// SIMATIC STEP 7 (V5.x) project PRACTICAS MOV-E
// CPU: CPU313 C-2 DP(1)
// station: P_ADR_BUS
// station: Hardware
// station: Equipo SIMATIC 300
// program: Programa S7(1)

SYMBOL_TABLE
"FLANCOS"	DB 1	DB 1
"P MARCHA"	I 0.0	BOOL
"P PARO"	I 0.1	BOOL
"Cycle Execution"	OB 1	OB 1
END_SYMBOL_TABLE

DATA_BLOCK "FLANCOS"	// DB 1
VERSION : 0.1
  STRUCT
   M0 : BOOL ;
   M1 : BOOL ;
   M2 : BOOL ;
   M3 : BOOL ;
   M4 : BOOL ;
   M5 : BOOL ;
   M6 : BOOL ;
   M7 : BOOL ;
  END_STRUCT ;	
BEGIN
END_DATA_BLOCK

ORGANIZATION_BLOCK "Cycle Execution"	// OB 1
TITLE = "Main Program Sweep (Cycle)"
VERSION : 0.1
VAR_TEMP
  OB1_EV_CLASS : BYTE ;	//Bits 0-3 = 1 (Coming event), Bits 4-7 = 1 (Event class 1)
  OB1_SCAN_1 : BYTE ;	//1 (Cold restart scan 1 of OB 1), 3 (Scan 2-n of OB 1)
  OB1_PRIORITY : BYTE ;	//Priority of OB Execution
  OB1_OB_NUMBR : BYTE ;	//1 (Organization block 1, OB1)
  OB1_RESERVED_1 : BYTE ;	//Reserved for system
  OB1_RESERVED_2 : BYTE ;	//Reserved for system
  OB1_PREV_CYCLE : INT ;	//Cycle time of previous OB1 scan (milliseconds)
  OB1_MIN_CYCLE : INT ;	//Minimum cycle time of OB1 (milliseconds)
  OB1_MAX_CYCLE : INT ;	//Maximum cycle time of OB1 (milliseconds)
  OB1_DATE_TIME : DATE_AND_TIME ;	//Date and time OB1 started
END_VAR
BEGIN
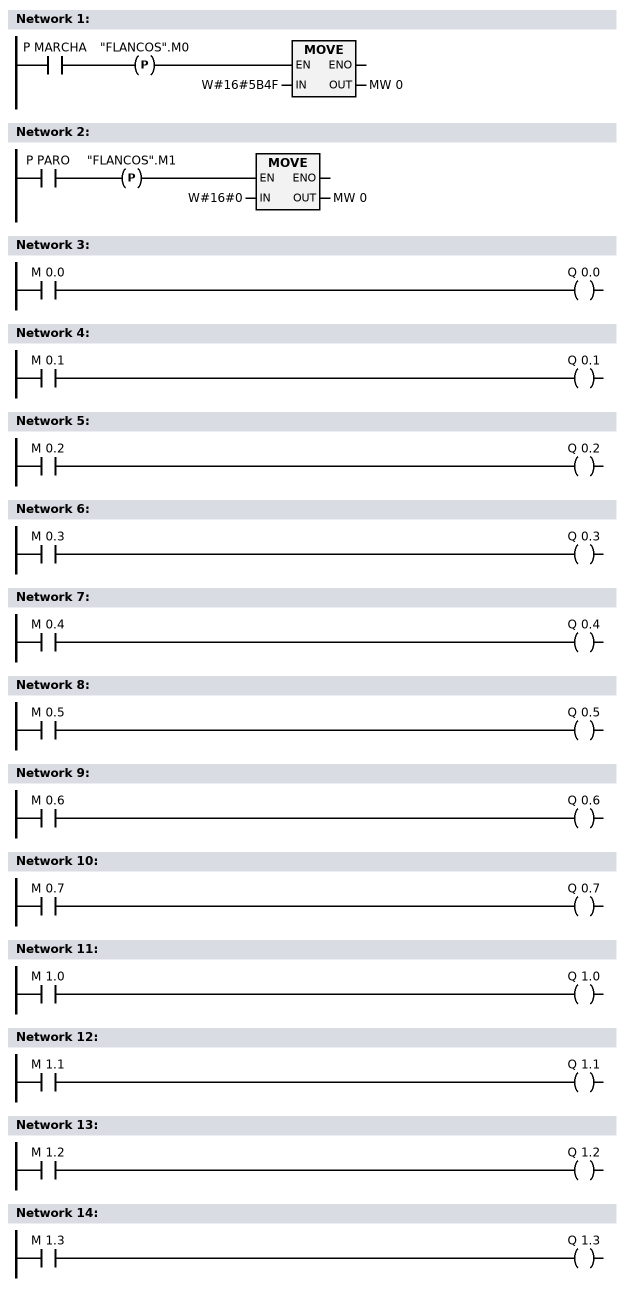
NETWORK
TITLE =
      A     "P MARCHA";
      FP    "FLANCOS".M0;
      JNB   _001;
      L     W#16#5B4F;
      T     MW 0;
_001: NOP   0;
NETWORK
TITLE =
      A     "P PARO";
      FP    "FLANCOS".M1;
      JNB   _002;
      L     W#16#0;
      T     MW 0;
_002: NOP   0;
NETWORK
TITLE =
      A     M 0.0;
      =     Q 0.0;
NETWORK
TITLE =
      A     M 0.1;
      =     Q 0.1;
NETWORK
TITLE =
      A     M 0.2;
      =     Q 0.2;
NETWORK
TITLE =
      A     M 0.3;
      =     Q 0.3;
NETWORK
TITLE =
      A     M 0.4;
      =     Q 0.4;
NETWORK
TITLE =
      A     M 0.5;
      =     Q 0.5;
NETWORK
TITLE =
      A     M 0.6;
      =     Q 0.6;
NETWORK
TITLE =
      A     M 0.7;
      =     Q 0.7;
NETWORK
TITLE =
      A     M 1.0;
      =     Q 1.0;
NETWORK
TITLE =
      A     M 1.1;
      =     Q 1.1;
NETWORK
TITLE =
      A     M 1.2;
      =     Q 1.2;
NETWORK
TITLE =
      A     M 1.3;
      =     Q 1.3;
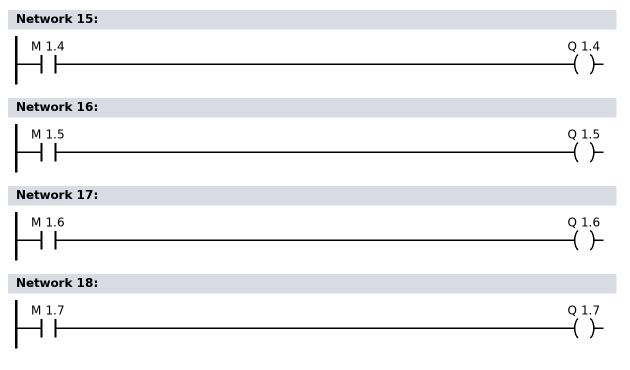
NETWORK
TITLE =
      A     M 1.4;
      =     Q 1.4;
NETWORK
TITLE =
      A     M 1.5;
      =     Q 1.5;
NETWORK
TITLE =
      A     M 1.6;
      =     Q 1.6;
NETWORK
TITLE =
      A     M 1.7;
      =     Q 1.7;
END_ORGANIZATION_BLOCK
